Staubli VAL3: AxisIsNeg.pgx

public program AxisIsNeg(bool x_b8Axis (dimensions=1), bool& x_bRes (dimensions=1))
begin
  x_bRes=false

  if x_b8Axis
    x_bRes=aioGet(aAio["In4_a8CurPosH"])>=3000

  else

    x_bRes=aioGet(aAio["In4_a7CurPosH"])>=3000

  endIf





end
